PROGRAM POU
VAR
	error: UINT;
	TempPID: FB_BasicPID;
	test: BOOL;

END_VAR

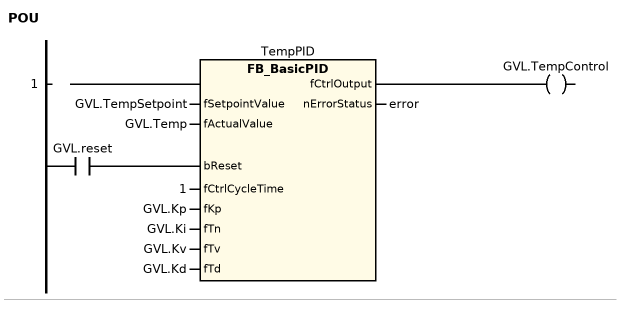
// NETWORK 1
TempPID(
    fSetpointValue := GVL.TempSetpoint,
    fActualValue := GVL.Temp,
    bReset := GVL.reset,
    fCtrlCycleTime := 1,
    fKp := GVL.Kp,
    fTn := GVL.Ki,
    fTv := GVL.Kv,
    fTd := GVL.Kd,
    nErrorStatus => error); // FB_BasicPID
GVL.TempControl := TempPID.fCtrlOutput;

END_PROGRAM

(* stored: Version 1.1.0.1, ProductVersion 3.1.4022.18
   POU POU: Id {3231294a-09f5-4b2a-98bd-60925c5024a2}, SpecialFunc None *)
